KUKA KRL program: coger.src, coger.dat

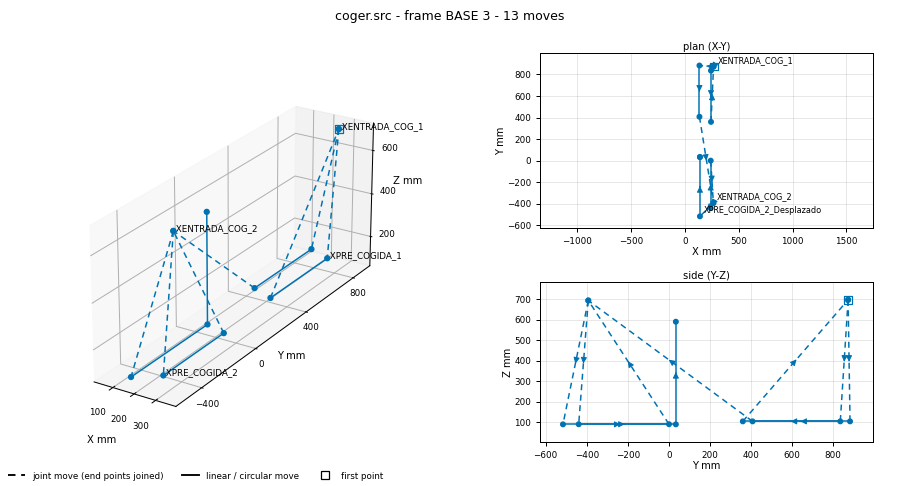
[picture p0: tool path of coger.src in frame BASE 3, 13 of 13 moves have a stored position in this frame; points joined in program order, loops and branches not executed]
--- coger.src ---
&ACCESS RVO1
&REL 60
&PARAM TEMPLATE = C:\KRC\Roboter\Template\vorgabe
&PARAM EDITMASK = *
DEF coger( )


;FOLD INI
  ;FOLD BASISTECH INI
    GLOBAL INTERRUPT DECL 3 WHEN $STOPMESS==TRUE DO IR_STOPM ( )
    INTERRUPT ON 3
    BAS (#INITMOV,0 )
  ;ENDFOLD (BASISTECH INI)
  ;FOLD USER INI
    ;Make your modifications here

  ;ENDFOLD (USER INI)
;ENDFOLD (INI)


IF (not GARRAS_CERRADAS) THEN

    PULSE (CERRAR_GARRAS,TRUE,0.5)

ENDIF



SWITCH TIPO_COGIDA

CASE 1 ;COGIDA 1

;FOLD PTP ENTRADA_COG_1 Vel=100 % PDAT1 Tool[2]:MORDAZA Base[3]:TRANSPORTADOR;%{PE}%R 5.6.16,%MKUKATPBASIS,%CMOVE,%VPTP,%P 1:PTP, 2:ENTRADA_COG_1, 3:, 5:100, 7:PDAT1
$BWDSTART=FALSE
PDAT_ACT=PPDAT1
FDAT_ACT=FENTRADA_COG_1
BAS(#PTP_PARAMS,100)
PTP XENTRADA_COG_1
;ENDFOLD



  ;FOLD PTP PRE_COGIDA_1 Vel=100 % PDAT4 Tool[2]:MORDAZA Base[3]:TRANSPORTADOR;%{PE}%R 5.6.16,%MKUKATPBASIS,%CMOVE,%VPTP,%P 1:PTP, 2:PRE_COGIDA_1, 3:, 5:100, 7:PDAT4
  $BWDSTART=FALSE
  PDAT_ACT=PPDAT1
  FDAT_ACT=FPRE_COGIDA_1
  BAS(#PTP_PARAMS,100)
  PTP XPRE_COGIDA_1
  ;ENDFOLD


LIN_REL {Y -475} C_DIS


CASE 2 ;COGIDA 1 DESPLAZADA

  ;FOLD PTP ENTRADA_COG_1 Vel=100 % PDAT1 Tool[2]:MORDAZA Base[3]:TRANSPORTADOR;%{PE}%R 5.6.16,%MKUKATPBASIS,%CMOVE,%VPTP,%P 1:PTP, 2:ENTRADA_COG_1, 3:, 5:100, 7:PDAT1
  $BWDSTART=FALSE
  PDAT_ACT=PPDAT1
  FDAT_ACT=FENTRADA_COG_1
  BAS(#PTP_PARAMS,100)
  PTP XENTRADA_COG_1
  ;ENDFOLD

  ;FOLD PTP PRE_COGIDA_1_Desplazado Vel=100 % PDAT4 Tool[2]:MORDAZA Base[3]:TRANSPORTADOR;%{PE}%R 5.6.16,%MKUKATPBASIS,%CMOVE,%VPTP,%P 1:PTP, 2:PRE_COGIDA_1, 3:, 5:100, 7:PDAT4
  $BWDSTART=FALSE
  PDAT_ACT=PPDAT1
  FDAT_ACT=FPRE_COGIDA_1_Desplazado
  BAS(#PTP_PARAMS,100)
  PTP XPRE_COGIDA_1_Desplazado
  ;ENDFOLD

  LIN_REL {Y -475} C_DIS

CASE 3 ;COGIDA 2
  ;FOLD PTP ENTRADA_COG_2 Vel=100 % PDAT2 Tool[2]:MORDAZA Base[3]:TRANSPORTADOR;%{PE}%R 5.6.16,%MKUKATPBASIS,%CMOVE,%VPTP,%P 1:PTP, 2:ENTRADA_COG_2, 3:, 5:100, 7:PDAT2
  $BWDSTART=FALSE
  PDAT_ACT=PPDAT1
  FDAT_ACT=FENTRADA_COG_2
  BAS(#PTP_PARAMS,100)
  PTP XENTRADA_COG_2
  ;ENDFOLD


  ;FOLD PTP PRE_COGIDA_2 Vel=100 % PDAT3 Tool[2]:MORDAZA Base[3]:TRANSPORTADOR;%{PE}%R 5.6.16,%MKUKATPBASIS,%CMOVE,%VPTP,%P 1:PTP, 2:PRE_COGIDA_2, 3:, 5:100, 7:PDAT3
  $BWDSTART=FALSE
  PDAT_ACT=PPDAT1
  FDAT_ACT=FPRE_COGIDA_2
  BAS(#PTP_PARAMS,100)
  PTP XPRE_COGIDA_2
  ;ENDFOLD


  LIN_REL {Y +440} C_DIS



CASE 4 ;COGIDA 2 DESPLAZADA



  ;FOLD PTP ENTRADA_COG_2 Vel=100 % PDAT2 Tool[2]:MORDAZA Base[3]:TRANSPORTADOR;%{PE}%R 5.6.16,%MKUKATPBASIS,%CMOVE,%VPTP,%P 1:PTP, 2:ENTRADA_COG_2, 3:, 5:100, 7:PDAT2
  $BWDSTART=FALSE
  PDAT_ACT=PPDAT1
  FDAT_ACT=FENTRADA_COG_2
  BAS(#PTP_PARAMS,100)
  PTP XENTRADA_COG_2
  ;ENDFOLD


  ;FOLD PTP FPRE_COGIDA_2_Desplazado Vel=100 % PDAT3 Tool[2]:MORDAZA Base[3]:TRANSPORTADOR;%{PE}%R 5.6.16,%MKUKATPBASIS,%CMOVE,%VPTP,%P 1:PTP, 2:PRE_COGIDA_2, 3:, 5:100, 7:PDAT3
  $BWDSTART=FALSE
  PDAT_ACT=PPDAT1
  FDAT_ACT=FPRE_COGIDA_2_Desplazado
  BAS(#PTP_PARAMS,100)
  PTP XPRE_COGIDA_2_Desplazado
  ;ENDFOLD

  LIN_REL {Y 550} C_DIS


ENDSWITCH


EXTENDER_PISADORES=TRUE

WAIT SEC 0.3 ;A falta de confirmacion de que PISADORES_EXTENDIDOS


LIN_REL {Z 500} C_DIS

;LE DIGO AL PLC QUE YA HE COGIDO SACO DE T1
PULSE (SACO_COGIDO_T1,TRUE,0.5)



          IF NOT LIMITE_CAPAS_DARSENA1 THEN

                 DEJAR_DARSENA1()

          ELSE
                  DEJAR_DARSENA2()
          ENDIF

          ;IF (NOT PRODUCCION_MIXTA AND PERMISO_DEJAR_DARSENA2)
;           DEJAR_DARSENA2()
          ;ENDIF


END

--- coger.dat ---
&ACCESS RVO1
&REL 60
&PARAM TEMPLATE = C:\KRC\Roboter\Template\vorgabe
&PARAM EDITMASK = *
DEFDAT  COGER
;FOLD EXTERNAL DECLARATIONS;%{PE}%MKUKATPBASIS,%CEXT,%VCOMMON,%P
;FOLD BASISTECH EXT;%{PE}%MKUKATPBASIS,%CEXT,%VEXT,%P
EXT  BAS (BAS_COMMAND  :IN,REAL  :IN )
DECL INT SUCCESS
;ENDFOLD (BASISTECH EXT)
;FOLD USER EXT;%{E}%MKUKATPUSER,%CEXT,%VEXT,%P
;Make here your modifications

;ENDFOLD (USER EXT)
;ENDFOLD (EXTERNAL DECLARATIONS)



DECL E6POS XENTRADA_COG_2={X 265.496094,Y -392.578308,Z 692.825317,A -179.405304,B -0.699936926,C 177.584,S 6,T 58,E1 0.0,E2 0.0,E3 0.0,E4 0.0,E5 0.0,E6 0.0}
DECL FDAT FENTRADA_COG_2={TOOL_NO 2,BASE_NO 3,IPO_FRAME #BASE,POINT2[] " ",TQ_STATE FALSE}

DECL E6POS XPRE_COGIDA_2={X 240.926605,Y -439.278015,Z 89.8367691,A -179.406006,B -0.698881328,C 177.583603,S 6,T 58,E1 0.0,E2 0.0,E3 0.0,E4 0.0,E5 0.0,E6 0.0}
DECL FDAT FPRE_COGIDA_2={TOOL_NO 2,BASE_NO 3,IPO_FRAME #BASE,POINT2[] " ",TQ_STATE FALSE}

DECL E6POS XCOGIDA_2={X 243.030304,Y 106.146301,Z 97.9635696,A -179.409698,B -0.447008699,C 177.583603,S 6,T 59,E1 0.0,E2 0.0,E3 0.0,E4 0.0,E5 0.0,E6 0.0}
DECL FDAT FCOGIDA_2={TOOL_NO 2,BASE_NO 3,IPO_FRAME #BASE,POINT2[] " ",TQ_STATE FALSE}

DECL E6POS XPRE_COGIDA_2_Desplazado={X 140.906494,Y -515.904785,Z 89.2991791,A -179.406601,B -0.701284826,C 177.582703,S 6,T 58,E1 0.0,E2 0.0,E3 0.0,E4 0.0,E5 0.0,E6 0.0}
DECL FDAT FPRE_COGIDA_2_Desplazado={TOOL_NO 2,BASE_NO 3,IPO_FRAME #BASE,POINT2[] " ",TQ_STATE FALSE}

DECL E6POS XENTRADA_COG_1={X 267.286011,Y 873.432312,Z 696.154785,A 1.04446101,B 1.65242505,C 179.309204,S 6,T 59,E1 0.0,E2 0.0,E3 0.0,E4 0.0,E5 0.0,E6 0.0}
DECL FDAT FENTRADA_COG_1={TOOL_NO 2,BASE_NO 3,IPO_FRAME #BASE,POINT2[] " ",TQ_STATE FALSE}

DECL E6POS XPRE_COGIDA_1={X 243.595703,Y 835.349121,Z 103.8489,A 0.0495731011,B 0.864072084,C 179.297302,S 6,T 59,E1 0.0,E2 0.0,E3 0.0,E4 0.0,E5 0.0,E6 0.0}
DECL FDAT FPRE_COGIDA_1={TOOL_NO 2,BASE_NO 3,IPO_FRAME #BASE,POINT2[] " ",TQ_STATE FALSE}

DECL E6POS XCOGIDA_1={X 248.395905,Y 356.371399,Z 96.664299,A 0.0506648198,B 0.865561903,C 179.296402,S 6,T 59,E1 0.0,E2 0.0,E3 0.0,E4 0.0,E5 0.0,E6 0.0}
DECL FDAT FCOGIDA_1={TOOL_NO 2,BASE_NO 3,IPO_FRAME #BASE,POINT2[] " ",TQ_STATE FALSE}


DECL E6POS XPRE_COGIDA_1_Desplazado={X 136.471603,Y 882.782288,Z 103.830803,A 0.0496506989,B 0.863984823,C 179.297394,S 6,T 59,E1 0.0,E2 0.0,E3 0.0,E4 0.0,E5 0.0,E6 0.0}
DECL FDAT FPRE_COGIDA_1_Desplazado={TOOL_NO 2,BASE_NO 3,IPO_FRAME #BASE,POINT2[] " ",TQ_STATE FALSE}



DECL PDAT PPDAT1={VEL 100.0,ACC 100.0,APO_DIST 100.0}
DECL LDAT LCPDAT1={VEL 2.0,ACC 100.0,APO_DIST 100.0,APO_FAC 50.0,ORI_TYP #VAR,CIRC_TYP #BASE,JERK_FAC 50.0,EXAX_IGN 0}

DECL BASIS_SUGG_T LAST_BASIS={POINT1[] "P0                      ",POINT2[] "P0                      ",CP_PARAMS[] "CPDAT0                  ",PTP_PARAMS[] "PDAT0                   ",CONT[] "                        ",CP_VEL[] "2.0                     ",PTP_VEL[] " 100                    ",SYNC_PARAMS[] "SYNCDAT                 ",SPL_NAME[] "S0                      "}
ENDDAT
